// Mitsubishi GX Works2 project: PART2   PLC: FX3G

// global labels: Global1
VAR_GLOBAL
  X_10 AT X010 : BOOL;
  Y_10 AT Y010 : BOOL;
  X_6 AT X006 : BOOL;
  X_2 AT X002 : BOOL;
  Y_2 AT Y002 : BOOL;
  Y_6 AT Y006 : BOOL;
  CC_1 AT CC1 : BOOL;
  CS_1 AT CS1 : BOOL;
  CS_2 AT CS2 : BOOL;
  CC_2 AT CC2 : BOOL;
END_VAR
VAR_GLOBAL CONSTANT
  sec_10 : INT := 100;
END_VAR
VAR_GLOBAL
  M_1 AT M1 : BOOL;
END_VAR
VAR_GLOBAL CONSTANT
  k_10 : INT := 10;
END_VAR
VAR_GLOBAL
  TC_5 AT TC5 : BOOL;
  TS_5 AT TS5 : BOOL;
  X_7 AT X007 : BOOL;
END_VAR

// task Task_01 (event TRUE, interval 0, priority 31): POU_01

PROGRAM POU_01
(* structured ladder/FBD written out as ST: instructions are called as NAME(EN, inputs, outputs); _pN, _eN, _tN stand for wires *)
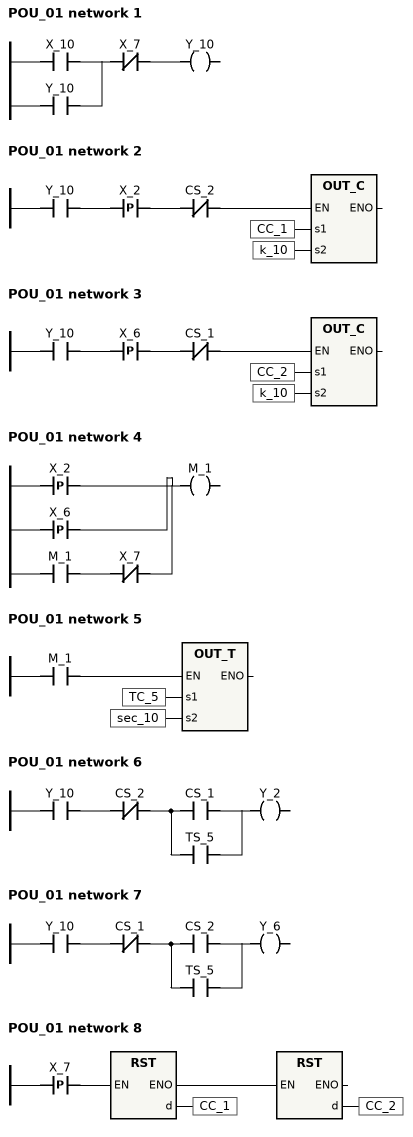
(* network 1 *)
Y_10 := (X_10 OR Y_10) AND NOT X_7;
(* network 2 *)
OUT_C(Y_10 AND LDP(TRUE, X_2) AND NOT CS_2, CC_1, k_10);
(* network 3 *)
OUT_C(Y_10 AND LDP(TRUE, X_6) AND NOT CS_1, CC_2, k_10);
(* network 4 *)
M_1 := LDP(TRUE, X_2) OR LDP(TRUE, X_6) OR (M_1 AND NOT X_7);
(* network 5 *)
OUT_T(M_1, TC_5, sec_10);
(* network 6 *)
_p1 := Y_10 AND NOT CS_2;
Y_2 := (_p1 AND CS_1) OR (_p1 AND TS_5);
(* network 7 *)
_p1 := Y_10 AND NOT CS_1;
Y_6 := (_p1 AND CS_2) OR (_p1 AND TS_5);
(* network 8 *)
_e1 := RST(LDP(TRUE, X_7), CC_1);
RST(_e1, CC_2);
END_PROGRAM
